(* CODESYS project CtaAppBmk_2.0.0.1.library
   Description: Bmk Library der CTA
   Version: 2.0.0.1
   Title: CtaAppBmk
   Author: SIS
   DocFormat: reStructuredText
   LanguageModelAttribute: qualified-access-only
   Placeholder: CtaAppBmk
   DefaultNamespace: CtaAppBmk
   CompiledLibraryCompatibilityVersion: CODESYS V3.5 SP20 Patch 5
   Company: CTA

Project tree, tasks and I/O mapping:
  libraries: CtaSysBase, 1.0.0.0 (CTA); TextListUtils, 4.5.0.0 (System); CtaVisSymbols, 2.0.0.0 (CTA); VisuSymbols, 4.5.0.0 (System); CtaVisApps, 1.0.0.0 (CTA); CtaVisHelp, 2.0.0.0 (CTA); CtaVisUser, 1.0.0.0 (CTA); CmpDynamicText, 3.5.20.0 (System)
  40 Visualizations/
    visualisation visObjInfoIntern
    visualisation visObjInfo
  30 Program Organization Units/
    function block fbBMK [ST]: proGetBMK, proGetAKS, proGetVendorDesignation, proGetCustomerDesignation, proGetObjectId, proNoBmkInList
  00000000-0000-0000-0000-000000000000|D:\CoDeSys\LibrariesV3\trunk\Intern\CAA\CAA Template\3.4.0.0 draft\Placeholder.xml
  00000000-0000-0000-0000-000000000000|D:\CoDeSys\LibrariesV3\trunk\Intern\CAA\CAA Template\3.2.0.3 draft\Prefix.pdf
  00000000-0000-0000-0000-000000000000|D:\CoDeSys\LibrariesV3\trunk\Intern\CAA\CAA Template\3.5.2.0 draft\Placeholder.xml
  20 Structs/
  50 Images/
  10 Documenation/
    global variables VersionHistory
    global variables readMe
  21 Interface/
    interface ITF_BMK: proGetAKS, proGetBMK, proGetObjectId, proNoBmkInList, proGetCustomerDesignation, proGetVendorDesignation
  11 Library Parameter/
    global variables Parameter
  12 Konstanten/
  60 Textlisten/
  13 Globale Variablen/
  text list GlobalTextList
*)

// 10 Documenation/VersionHistory
(* 

.. image:: ../../Images/CTA_Logo.jpg
   :align: right
   :width: 15% 

**Vorlage**   


============ =========== =========== ============================================
**Date**     **Version** **Author**  **Change**
------------ ----------- ----------- --------------------------------------------
04.03.2021   0.0.0.0     SIS         Vorlage erstellt

============ =========== =========== ============================================


*)
VAR_GLOBAL
    stInfo : STRING:= '0.0.0.0, Vorlage, CTA';
END_VAR

// 10 Documenation/readMe
(*

**ReadMe**
 
 |	**Empfehlung**
 |
 |	Dokumentrieren Sie die Library für eine nachhaltige Entwicklung
 |     
 | *Beispiel* 
 |
 | Dies ist die Vorlage Library der CTA. Erstellen Sie ihre Library anhand dieser Vorlage.
*)

VAR_GLOBAL
    xReadMeDone              :   BOOL;
END_VAR

// 11 Library Parameter/Parameter
{attribute 'qualified_only' := ''}
VAR_GLOBAL CONSTANT
	stTextListBmk					: STRING := 'BMK';
	stTextListAks					: STRING := 'AKS';
	stTextListVendorDesignation		: STRING := 'VendorDesignation';
	stTextListCustomerDesignation	: STRING := 'CustomerDesignation';
END_VAR

// 30 Program Organization Units/fbBMK
(* BMK Functionblock single Responsibility operating resources indicator BMK *)
{attribute 'enable_dynamic_creation'}
FUNCTION_BLOCK fbBMK EXTENDS CtaSysBase.fbBASE IMPLEMENTS ITF_BMK
VAR_INPUT
	/// Object ID
	{attribute 'monitoring_encoding' := 'UTF-8'}
	stObjId: STRING(20);
END_VAR
VAR
	/// Flag no BMK in List
	xNoBmkInList: BOOL;
END_VAR

{IF NOT defined (task:VISU_TASK) AND (defined (task:PLC_Task) OR defined (resource:Steuerung))}
    {error 'No VisualizationManager or No VISU_TASK in Application'}  
{END_IF}

{attribute 'monitoring':='call'}
{attribute 'monitoring_encoding' := 'UTF-8'}
PROPERTY proGetBMK : STRING(7)
GET
VAR
	pTempGetBmk		:	POINTER TO STRING(7);	
END_VAR
proGetBMK := '';
IF stObjId <> '' THEN
	(*Language dependent text*)
	__TRY
			pTempGetBmk := TLU.DynamicTextGetDefaultText(ADR(Parameter.stTextListBmk),ADR(stObjId));
			IF pTempGetBmk <> 0 THEN
				proGetBMK := pTempGetBmk^;
			END_IF;
	__CATCH
		proGetBMK := '';
	__ENDTRY
	(* Set xNoBmkInList if no BMK is found*)
	IF proGetBMK = '' THEN
		xNoBmkInList := TRUE;
        proGetBMK    := '-';
	ELSE
		xNoBmkInList := FALSE;
	END_IF;
ELSE
    proGetBMK    := '-';    
END_IF;
END_GET
END_PROPERTY

{attribute 'monitoring':='call'}
{attribute 'monitoring_encoding' := 'UTF-8'}
PROPERTY proGetAKS : STRING(40)
GET
proGetAKS := '';
IF stObjId <> '' THEN
	(*Language dependent text*)
	__TRY	
		TLU.GetText(Parameter.stTextListAks,stObjId,ADR(proGetAKS),SIZEOF(proGetAKS));
	__CATCH
		proGetAKS := '';
	__ENDTRY
END_IF;
END_GET
END_PROPERTY

{attribute 'monitoring':='call'}
{attribute 'monitoring_encoding' := 'UTF-8'}
PROPERTY proGetVendorDesignation : STRING(140)
GET
proGetVendorDesignation := '';
IF stObjId <> '' THEN
	(*Language dependent text*)
	__TRY
		TLU.GetText(Parameter.stTextListVendorDesignation,stObjId,ADR(proGetVendorDesignation),SIZEOF(proGetVendorDesignation)); 
	__CATCH
		TLU.CmpDynamicText.DynamicTextReloadTexts();
		proGetVendorDesignation := '';			
	__ENDTRY	
    IF proGetVendorDesignation = '' THEN
        proGetVendorDesignation := proGetInstancePath;
	END_IF;
ELSE
    proGetVendorDesignation := proGetInstancePath;    
END_IF;
END_GET
END_PROPERTY

{attribute 'monitoring':='call'}
{attribute 'monitoring_encoding' := 'UTF-8'}
PROPERTY proGetCustomerDesignation : STRING(100)
GET
VAR
    dwState :   DWORD;
END_VAR
proGetCustomerDesignation := '';
IF stObjId <> '' THEN
	(*Language dependent text*)
	__TRY
		dwState := TLU.GetText(Parameter.stTextListCustomerDesignation,stObjId,ADR(proGetCustomerDesignation),SIZEOF(proGetCustomerDesignation));
	__CATCH
		proGetCustomerDesignation := '';
	__ENDTRY	
END_IF;
END_GET
END_PROPERTY

{attribute 'monitoring':='call'}
{attribute 'monitoring_encoding' := 'UTF-8'}
PROPERTY proGetObjectId : STRING(20)
GET
proGetObjectId := stObjId;
END_GET
END_PROPERTY

{attribute 'monitoring':='call'}
{attribute 'monitoring_encoding' := 'UTF-8'}
PROPERTY proNoBmkInList : BOOL
GET
VAR
	stTestBMK :	STRING(7);
END_VAR
IF stObjId <> '' THEN
	(*Get state of xNoBmkInList*)
	stTestBMK := proGetBMK;
	proNoBmkInList := xNoBmkInList;
END_IF;
END_GET
END_PROPERTY

END_FUNCTION_BLOCK

// 21 Interface/ITF_BMK
/// BMK Interface single Responsibility operating resources indicator BMK
INTERFACE ITF_BMK EXTENDS CtaSysBase.ITF_BASE

{attribute 'monitoring':='call'}
PROPERTY proGetAKS : STRING(40)
GET
END_GET
END_PROPERTY

{attribute 'monitoring':='call'}
PROPERTY proGetBMK : STRING(7)
GET
END_GET
END_PROPERTY

{attribute 'monitoring':='call'}
PROPERTY proGetObjectId : STRING(20)
GET
END_GET
END_PROPERTY

{attribute 'monitoring':='call'}
PROPERTY proNoBmkInList : BOOL
GET
END_GET
END_PROPERTY

{attribute 'monitoring':='call'}
PROPERTY proGetCustomerDesignation : STRING(100)
GET
END_GET
END_PROPERTY

{attribute 'monitoring':='call'}
PROPERTY proGetVendorDesignation : STRING(140)
GET
END_GET
END_PROPERTY

END_INTERFACE

// 40 Visualizations/visObjInfoIntern
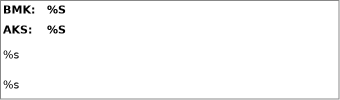
VISUALIZATION visObjInfoIntern  // 340x100
VAR_INPUT
	ITF_BMK_IN : ITF_BMK;
END_VAR
    Textfield (0,0 40x20), "BMK:"
    Textfield (0,20 40x20), "AKS:", invisible if: ITF_BMK_IN.proGetAKS = ''
    Textfield (40,0 300x20), "%S", text variable: SEL(ITF_BMK_IN.proNoBmkInList,ITF_BMK_IN.proGetBMK,'No BMK Found')
    Textfield (40,20 300x20), "%S", text variable: ITF_BMK_IN.proGetAKS, invisible if: ITF_BMK_IN.proGetAKS = ''
    Textfield (0,40 340x30), "%s", tooltip "Hersteller Bezeichnung", text variable: ITF_BMK_IN.proGetVendorDesignation, invisible if: ITF_BMK_IN.proGetVendorDesignation = ''
    Textfield (0,70 340x30), "%s", tooltip "Kunden Bezeichnung", text variable: ITF_BMK_IN.proGetCustomerDesignation, invisible if: ITF_BMK_IN.proGetCustomerDesignation = ''
END_VISUALIZATION

// 40 Visualizations/visObjInfo
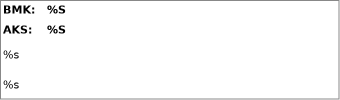
VISUALIZATION visObjInfo  // 340x100
VAR_INPUT
	ITF_BMK_IN : ITF_BMK;
END_VAR
    Frame (0,0 340x100), invisible if: ITF_BMK_IN =0
        shows visObjInfoIntern(ITF_BMK_IN := ITF_BMK_IN)
END_VISUALIZATION
